ABB RobotStudio station: jaffir robot despensing.rsstn

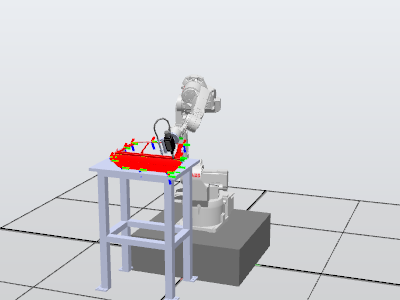
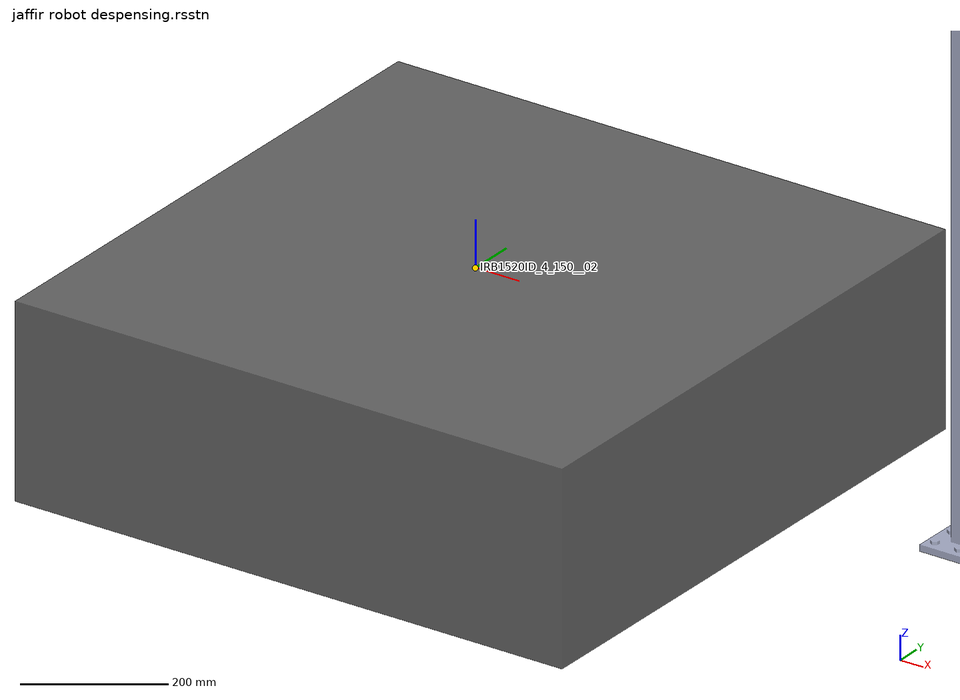
[picture v1: parts stored in the station drawn from their meshes, with robot base, taught points and paths (robot models come from the ABB library and are not in the file)]
Station Station (saved by RobotStudio 22.3.10141.1)
Controller Controller43, task T_ROB1: task frame (RAPID world) sits at (0, 0, 300) mm in the station
Controller Controller43
  mechanical unit ROB_1: IRB1520ID_4_150__02, 6 joints, base frame (0, 0, 0) mm
Layout (positions relative to the parent item):
  - IRB1520ID_4_150__02 [mechanism, from Robots\IRB1520ID_4_150_G_02.rslib] at (0, 0, 300) mm; joint values [0.2087, 0.0903, 0.1169, -0.5176, 0.371, 0.5933] (rad or m)
  - Part_3 [part] at (0, 10.65, 0) mm, size 900 x 900 x 300 mm
  - Dispencer [mechanism, from Dispencing\Dispencer.rslib] at (1114.2, 199.24, 1287.65) mm, rotated rx 180 ry 60 rz 180 deg
  - table with door_2 [part] at (1506.39, 276.46, 623.59) mm, rotated rx 90 ry 0 rz -90 deg, size 600 x 960.7 x 450 mm
Attachment: Dispencer is attached to IRB1520ID_4_150__02 / Link6
Targets, tools, work objects and paths stored in the station, written as RAPID:
! task T_ROB1
MODULE CalibData
  PERS tooldata Dispencer:=[TRUE,[[145,-0.097,55],[0.707106781,0,0.707106781,0]],[1,[0,0,1],[1,0,0,0],0,0,0]];
ENDMODULE

! task T_ROB1
MODULE Module1
  CONST robtarget Target_10:=[[928.998833175,201.544010962,900.133087705],[0.258819026,0,-0.965925831,0.000000005],[0,-1,0,0],[9E+09,9E+09,9E+09,9E+09,9E+09,9E+09]];
  CONST robtarget Target_20:=[[1083.063015043,239.989818398,848.198787075],[0.258819026,-0.000000001,-0.965925831,0],[0,-1,0,0],[9E+09,9E+09,9E+09,9E+09,9E+09,9E+09]];
  CONST robtarget Target_30:=[[1167.765990164,261.218494379,809.121631267],[0.258819021,-0.000000005,-0.965925833,-0.000000018],[0,-1,0,0],[9E+09,9E+09,9E+09,9E+09,9E+09,9E+09]];
  CONST robtarget Target_40:=[[1362.988024375,272.394388101,802.211284071],[0.258819028,-0.000000009,-0.965925831,-0.000000016],[0,-1,0,0],[9E+09,9E+09,9E+09,9E+09,9E+09,9E+09]];
  CONST robtarget Target_50:=[[919.237025051,85.687589145,903.423754846],[0.258819013,-0.000000013,-0.965925835,-0.000000023],[0,-1,0,0],[9E+09,9E+09,9E+09,9E+09,9E+09,9E+09]];
  CONST robtarget Target_60:=[[927.384384713,-29.926433089,900.677344459],[0.258819023,-0.000000013,-0.965925832,-0.000000021],[-1,0,-1,0],[9E+09,9E+09,9E+09,9E+09,9E+09,9E+09]];
  CONST robtarget Target_70:=[[972.354900696,-164.452699322,887.145903946],[0.258819014,-0.000000017,-0.965925835,-0.00000004],[-1,0,-1,0],[9E+09,9E+09,9E+09,9E+09,9E+09,9E+09]];
  CONST robtarget Target_80:=[[1030.72501063,-191.365103028,865.841701923],[0.258819024,-0.000000019,-0.965925832,-0.000000035],[-1,0,-1,0],[9E+09,9E+09,9E+09,9E+09,9E+09,9E+09]];
  CONST robtarget Target_90:=[[1123.193991434,-250.314012014,817.228401037],[0.258819019,-0.000000023,-0.965925833,-0.000000035],[-1,0,-1,0],[9E+09,9E+09,9E+09,9E+09,9E+09,9E+09]];
  CONST robtarget Target_100:=[[1177.381062367,-212.61299462,809.450406857],[0.258819014,-0.000000028,-0.965925835,-0.00000006],[-1,0,-1,0],[9E+09,9E+09,9E+09,9E+09,9E+09,9E+09]];
  CONST robtarget Target_110:=[[1326.903011997,-63.38147124,814.044190532],[0.258819017,-0.000000027,-0.965925834,-0.000000057],[-1,0,-1,0],[9E+09,9E+09,9E+09,9E+09,9E+09,9E+09]];
  CONST robtarget Target_120:=[[1354.52202307,73.33055434,822.338233719],[0.25881902,-0.000000027,-0.965925833,-0.000000058],[0,-1,0,0],[9E+09,9E+09,9E+09,9E+09,9E+09,9E+09]];
  CONST robtarget Target_130:=[[1341.037068053,255.105927824,817.923185314],[0.258819028,-0.000000021,-0.965925831,-0.00000005],[0,-1,0,0],[9E+09,9E+09,9E+09,9E+09,9E+09,9E+09]];
  CONST robtarget Target_140:=[[1274.445086896,266.560114256,803.2087262],[0.258819019,-0.000000017,-0.965925833,-0.000000053],[0,-1,0,0],[9E+09,9E+09,9E+09,9E+09,9E+09,9E+09]];
  CONST robtarget Target_150:=[[1089.33307165,-228.742791808,834.575422819],[0.258819027,-0.000000011,-0.965925831,-0.000000051],[-1,0,-1,0],[9E+09,9E+09,9E+09,9E+09,9E+09,9E+09]];
  CONST robtarget Target_160:=[[1089.33307316,-43.716402586,834.575440853],[0.258819014,-0.000000012,-0.965925835,-0.000000048],[-1,0,-1,0],[9E+09,9E+09,9E+09,9E+09,9E+09,9E+09]];
  CONST robtarget Target_170:=[[1089.333071153,199.14251351,834.57544163],[0.258819014,-0.000000013,-0.965925835,-0.000000064],[0,-1,0,0],[9E+09,9E+09,9E+09,9E+09,9E+09,9E+09]];
  PROC Path_10()
  ENDPROC
ENDMODULE

